ABB RobotStudio station: conveier tracking_assingment(2).rsstn

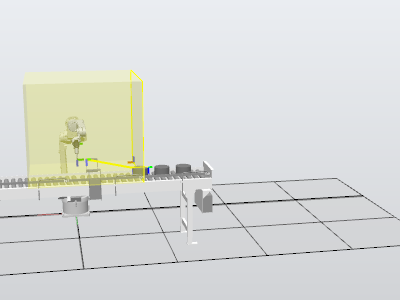
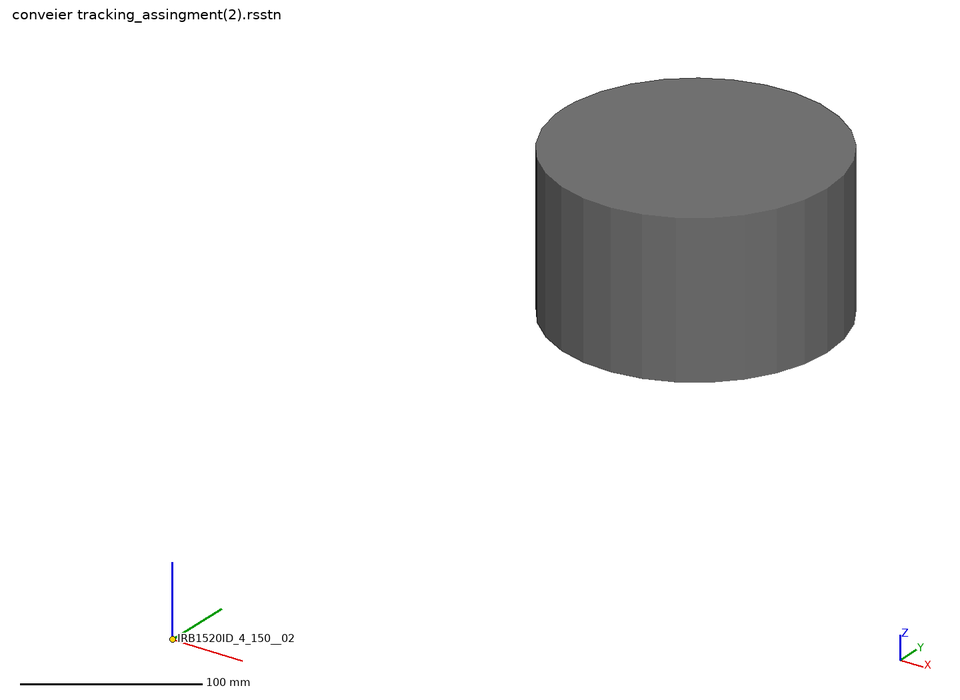
[picture v1: parts stored in the station drawn from their meshes, with robot base, taught points and paths (robot models come from the ABB library and are not in the file)]
Station conveier tracking_assingment(incomplet(error)) (saved by RobotStudio 22.3.10141.1)
Controller Controller29, task T_ROB1: task frame (RAPID world) sits at (-710.04, 543.58, 775) mm in the station
Controller Controller29
  mechanical unit ROB_1: IRB1520ID_4_150__02, 6 joints, base frame (710.04, -543.58, -775) mm, rotated rx 0 ry 0 rz 90 deg
  mechanical unit CNV1: ?, 1 joints, base frame (0, 500, 0) mm
Layout (positions relative to the parent item):
  - IRB1520ID_4_150__02 [mechanism, from Robots\IRB1520ID_4_150_G_02.rslib] at (0, 0, 0) mm, rotated rx 0 ry 0 rz 90 deg; joint values [0.7381, 0.5164, -0.4496, -0.9067, 0.8331, 1.1367] (rad or m)
  - MyTool [mechanism, from Training Objects\myTool.rslib] at (0, 1056.21, 1143) mm, rotated rx 180 ry 60 rz -90 deg
  - Conveyor [conveyor] at (0, 500, 0) mm
    - 400_guide [part] at (-1484.89, 541.08, 0) mm, size 3033 x 590 x 945 mm
    - Part_1 [part], size 176 x 175.7 x 100 mm
    - ConveyorObject_48 [conveyorobject] at (-704.44, 543.58, 775) mm
      - Part_1 [part] at (0, 190, 0) mm, size 176 x 175.7 x 100 mm
    - ConveyorObject_49 [conveyorobject] at (-954.44, 543.58, 775) mm
      - Part_1 [part] at (0, 190, 0) mm, size 176 x 175.7 x 100 mm
    - ConveyorObject_50 [conveyorobject] at (-1204.44, 543.58, 775) mm
      - Part_1 [part] at (0, 190, 0) mm, size 176 x 175.7 x 100 mm
Attachment: MyTool is attached to IRB1520ID_4_150__02 / Link6
Conveyor tracking Connection: unit CNV1, TravelOffset=0.7, QueueTrackDistance=0, StartWindowWidth=1.25, SyncSeparation=0.1, CountsPerMeter=10000
Collision set CollisionSet_1:  against , near miss 0 m
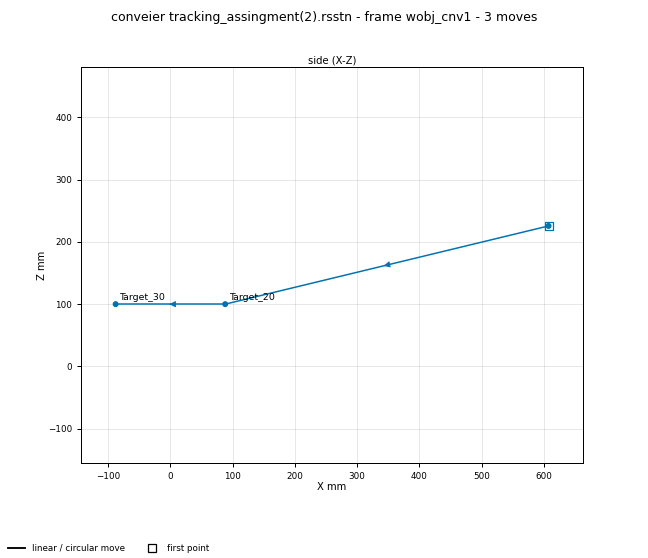
[picture p0: tool path of conveier tracking_assingment(2).rsstn in frame wobj_cnv1, 3 of 3 moves have a stored position in this frame; points joined in program order, loops and branches not executed]
Targets, tools, work objects and paths stored in the station, written as RAPID:
! task T_ROB1
MODULE CalibData
  PERS tooldata MyTool:=[TRUE,[[31.792631019,0,229.638935148],[0.945518576,0,0.325568154,0]],[1,[0,0,1],[1,0,0,0],0,0,0]];
  TASK PERS wobjdata wobj_cnv1:=[FALSE,FALSE,"CNV1",[[0,0,0],[1,0,0,0]],[[0,0,0],[1,0,0,0]]];
ENDMODULE

! task T_ROB1
MODULE Module1
  CONST robtarget Target_10:=[[607.494078146,195.60386714,225.64730631],[0.134922335,-0.694115238,0.694115238,0.134922335],[0,0,0,0],[9E+09,9E+09,9E+09,9E+09,9E+09,9E+09]];
  CONST robtarget Target_20:=[[87.999958619,189.999963087,99.999985507],[0.134922218,-0.694115251,0.694115268,0.13492223],[0,-1,0,0],[9E+09,9E+09,9E+09,9E+09,9E+09,0]];
  CONST robtarget Target_30:=[[-88.000024997,189.999985678,99.999997886],[0.134922151,-0.694115252,0.69411529,0.134922177],[0,-1,0,0],[9E+09,9E+09,9E+09,9E+09,9E+09,0]];
  PROC Path_10()
    MoveL Target_10,v1000,z100,MyTool\WObj:=wobj_cnv1;
    MoveL Target_20,v1000,z100,MyTool\WObj:=wobj_cnv1;
    MoveL Target_30,v1000,z100,MyTool\WObj:=wobj_cnv1;
  ENDPROC
ENDMODULE

